Staubli VAL3: _finish.pgx

program _finish()
begin
  // ============================================================================
  // CMD 1: 종료 - 홈 위치 복귀
  // ============================================================================
  cls()
  putln("[CMD 1] 종료 - 홈 복귀")
  nStatusSignal = 0

  movej(j_home, tTool, mNomSpeed)
  waitEndMove()

  putln("[CMD 1] 완료")
  bRunning = false

end
